PROGRAM MES_Controller
VAR
END_VAR

IF G_xComProtocol THEN
	OPCUA_Controller();
ELSE
	LOCAL_COM_Controller();
END_IF

END_PROGRAM

(* stored: Version 1.1.0.1, ProductVersion 3.1.4022.18
   POU MES_Controller: Id {68dc098d-b5d8-4165-929f-a366b3e946c8}, SpecialFunc None *)
